(* IEC 61131-3 sources: eCockpitGit/test_project/src/%F%00 Library/%F%Common Functions/%F%Networking/%POU%FB_TCPController, 6 files *)

(* ---- %METH%acceptConnection.st ---- *)
//Called to accept tcp connection
// |**Version**|**Author**| **Date** |**Changes**
// | 1         | NSN      | 20-05-22 | Creation
METHOD acceptConnection : BOOL
VAR_IN_OUT
	listener			:TCP.Listener;
END_VAR
VAR
	tcpError			:TCP.ERROR;
END_VAR
(*%!%__DELIMITER__%!%*)
IF NOT(S_open) THEN
	IF listener.Accept(pStream:=ADR(S_stream)) = TCP.ERROR.NO_ERROR THEN
		S_open					:=		TRUE;
		acceptConnection		:=		TRUE;
		IF S_management <> 0 THEN
			S_management.onOpen(index:=S_index,controller:=THIS^);
		END_IF
	END_IF
END_IF

(* ---- %METH%closeConnection.st ---- *)
//Called to close and clean up connection
// |**Version**|**Author**| **Date** |**Changes**
// | 1         | NSN      | 20-05-22 | Creation
METHOD closeConnection
(*%!%__DELIMITER__%!%*)
S_stream.Close();
S_stream.Reset();
S_open			:=		FALSE;
IF S_management <> 0 THEN
	S_management.onClose(index:=S_index,controller:=THIS^);
END_IF

(* ---- %METH%cycle.st ---- *)
//Called cyclicly
// |**Version**|**Author**| **Date** |**Changes**
// | 1         | NSN      | 20-05-22 | Creation
METHOD cycle
VAR
	i			:DINT;
	sent		:DINT;
	state		:TCP.STREAM_STATE;
END_VAR
(*%!%__DELIMITER__%!%*)
IF S_open THEN
	S_messageAmount							:=		0;
	IF S_sendAmount > 0 THEN
		CASE S_stream.Send(pbyBuffer:=S_sendBuffer,diBufferSize:=S_sendBufferSize,diSent=>sent) OF
			TCP.ERROR.NO_ERROR,TCP.ERROR.PENDING:
				IF S_sendAmount > sent THEN
					FOR i := 0 TO S_sendAmount - sent - 1 DO
						S_sendBuffer^[i]	:=		S_sendBuffer^[i + sent];
					END_FOR
					S_sendAmount			:=		S_sendAmount - sent;
				ELSE
					S_sendAmount			:=		0;
				END_IF
		ELSE
			closeConnection();
		END_CASE
	END_IF
END_IF

(* ---- %METH%initialize.st ---- *)
//Initializes the tcp controller with needed values
// |**Version**|**Author**| **Date** |**Changes**
// | 1         | NSN      | 20-05-22 | Creation
METHOD initialize : SLMResult
VAR_INPUT
	recieveBuffer		:POINTER TO ARRAY[0..99] OF BYTE;	//Reference to recieve buffer
	recieveBufferSize	:DINT;								//Size of recieve buffer
	sendBuffer			:POINTER TO ARRAY[0..99] OF BYTE;	//Reference to send buffer
	sendBufferSize		:DINT;								//Size of send buffer
	sendMaxSize			:DINT;								//Estimated max size of sending message, this makes sure that recieved messages are only processed when there is enough space to send the response in the send buffer
	maxMessages			:DINT;								//Limit for how many messages can be decoded per cycle
	headerSize			:DINT;								//Size of header for tcp message, reading wait until there is at least this amount in the buffer before decoding is performed
END_VAR

(*%!%__DELIMITER__%!%*)
IF recieveBuffer = 0 OR recieveBufferSize = 0 OR sendBuffer = 0 OR sendBufferSize = 0 THEN
	initialize.success	:=		FALSE;
	initialize.code		:=		ERCodes.FB_TCPController_initialize;
	RETURN;
END_IF
S_recieveBuffer			:=		recieveBuffer;
S_recieveBufferSize		:=		recieveBufferSize;
S_sendBuffer			:=		sendBuffer;
S_sendBufferSize		:=		sendBufferSize;
S_sendMaxSize			:=		sendMaxSize;
IF maxMessages = 0 THEN
	S_maxMessages		:=		1000;
ELSE
	S_maxMessages		:=		maxMessages;
END_IF
S_headerSize			:=		headerSize;

(* ---- %METH%readAmount.st ---- *)
//Called after data is read from read buffer, with amount read
// |**Version**|**Author**| **Date** |**Changes**
// | 1         | NSN      | 20-05-22 | Creation
METHOD readAmount : BOOL
VAR_INPUT
	amount			:DINT;
END_VAR
VAR
	i				:DINT;
END_VAR
(*%!%__DELIMITER__%!%*)
IF amount < S_recieveAmount THEN
	FOR i := 0 TO S_recieveAmount - amount - 1 DO
		S_recieveBuffer^[i]		:=		S_recieveBuffer^[i + amount];
	END_FOR
	S_recieveAmount				:=		S_recieveAmount - amount;
ELSE
	S_recieveAmount				:=		0;
END_IF

(* ---- %METH%sendData.st ---- *)
//Called to load data into send buffer
// |**Version**|**Author**| **Date** |**Changes**
// | 1         | NSN      | 20-05-22 | Creation
METHOD sendData : BOOL
VAR_INPUT
	data		:POINTER TO BYTE;
	size		:DINT;
END_VAR
VAR
	i			:DINT;
	sent		:DINT;
	remaining	:DINT;
END_VAR

(*%!%__DELIMITER__%!%*)
//If there is space in the send buffer
IF S_sendBufferSize - S_sendAmount >= size THEN
	IF S_sendAmount > 0 THEN
		FOR i := 0 TO size - 1 DO
			S_sendBuffer^[i + S_sendAmount]			:=		data[i];
		END_FOR
		S_sendAmount								:=		size;
	ELSE
		CASE S_stream.Send(pbyBuffer:=data,diBufferSize:=size,diSent=>sent) OF
			TCP.ERROR.NO_ERROR,TCP.ERROR.PENDING:
				IF size > sent THEN
					remaining							:=		size - sent;
					FOR i := 0 TO remaining - 1 DO
						S_sendBuffer^[i + S_sendAmount]	:=		data[i];
					END_FOR
					S_sendAmount						:=		S_sendAmount + remaining;
				END_IF
		ELSE
			closeConnection();
		END_CASE
	END_IF
END_IF
